(* IEC 61131-3 sources: RL_MAR/experiments/comparison/autoplc/results/gpt-4o_20260511_211137/hf_21, 1 file *)

(* ---- hf_21_3.st ---- *)
FUNCTION_BLOCK FB_SplitNumber
    VAR_INPUT
        InputNumber : INT;
    END_VAR

    VAR_OUTPUT
        Thousands : INT;
        Hundreds : INT;
        Tens : INT;
        Ones : INT;
        Min : INT;
        error : BOOL;
        status : WORD;
    END_VAR

    VAR
        tempNumber : INT;
        minValue : INT;
    END_VAR

    // Input Validation
    IF (InputNumber < 0) OR (InputNumber > 9999) THEN
        error := TRUE;
        status := 16#8001;
        Thousands := 0;
        Hundreds := 0;
        Tens := 0;
        Ones := 0;
        Min := 0;
    ELSE
        error := FALSE;
        status := 16#0000;

        // Digit Separation Logic
        Thousands := InputNumber / 1000;
        Hundreds := (InputNumber MOD 1000) / 100;
        Tens := (InputNumber MOD 100) / 10;
        Ones := InputNumber MOD 10;

        // Minimum Value Detection
        minValue := 32767; // Initialize to maximum possible INT value

        IF Thousands <> 0 THEN
            minValue := minimal(Thousands, minValue);
        END_IF;

        IF Hundreds <> 0 THEN
            minValue := minimal(Hundreds, minValue);
        END_IF;

        IF Tens <> 0 THEN
            minValue := minimal(Tens, minValue);
        END_IF;

        IF Ones <> 0 THEN
            minValue := minimal(Ones, minValue);
        END_IF;

        IF minValue = 32767 THEN
            Min := 0; // All digits are zero
        ELSE
            Min := minValue; // Found minimum non-zero digit
        END_IF;
    END_IF;
END_FUNCTION_BLOCK

FUNCTION minimal : INT
    VAR_INPUT
        IN1 : INT;
        IN2 : INT;
    END_VAR

    IF IN1 <= IN2 THEN
        minimal := IN1;
    ELSE
        minimal := IN2;
    END_IF;
END_FUNCTION
